{attribute 'qualified_only'}
VAR_GLOBAL
END_VAR

(* stored: Version 1.1.0.1, ProductVersion 3.1.4024.16
   GVL Global_1: Id {f32f36f6-8215-4998-8210-21d01fde39f9} *)
